// Implementation of a pseudo 3-way valve by controlling 2 outputs 
FUNCTION_BLOCK FV3
VAR_INPUT
	sp : BOOL := FALSE;
END_VAR
VAR_OUTPUT
	pv : BOOL := FALSE;
END_VAR
VAR
	passiveSV AT %Q*: BOOL;
	activeSV AT %Q*: BOOL;
END_VAR

passiveSV := NOT sp;
activeSV := sp;
pv := sp;

END_FUNCTION_BLOCK

(* stored: Version 1.1.0.1, ProductVersion 3.1.0.36
   POU FV3: Id {b569a884-7965-4230-9107-2f4d98e5e443}, SpecialFunc None *)
